FUNCTION_BLOCK PUBLIC ABSTRACT TcoKukaRoboticsTask EXTENDS TcoCore.TcoTask 
VAR_IN_OUT
    inoConfig 	: TcoKukaRobotics_Config_v_5_x_x;
	inoControl 	: TcoKukaRobotics_Control_v_5_x_x;
	inoStatus 	: TcoKukaRobotics_Status_v_5_x_x;	
END_VAR
VAR
	_errorMessage:TcoCore.TcoMessenger(THIS^);
    {attribute 'hide'} 
	_progress : INT := 0;
    {attribute 'hide'} 
	_infoTimer :  TON;
    {attribute 'hide'} 
	_errorTimer :  TON;
	{attribute 'hide'} 
	_timer :  TON;
    {attribute 'hide'} 
	_varInfo : __SYSTEM.VAR_INFO;
    {attribute 'hide'} 
	_sb : TcoCore.StringBuilder;
	{attribute 'hide'}
	_blink:TcoUtilities.TcoBlinker(THIS^);
END_VAR

METHOD CallTimers
VAR_INPUT
	inValue : BOOL;
END_VAR
IF  __ISVALIDREF(inoConfig) AND THIS^.inoConfig.ErrorTime <> T#0S OR NOT inValue THEN  
_errorTimer(IN := inValue, PT := THIS^.inoConfig.ErrorTime);
END_IF;
IF  __ISVALIDREF(inoConfig) AND THIS^.inoConfig.InfoTime <>T#0S OR NOT inValue THEN  
_infoTimer(IN := inValue, PT := THIS^.inoConfig.InfoTime);
END_IF;
END_METHOD

(*~
	<docu>
		<summary>
			Restores this instance to the Ready state. Can be called explicitly or from within one of the restore mechanisms.
			<para>
				See also <see cref="PlcDocu.TcoCore.TcoTask.AutoRestorable()"/>
			</para>
		</summary>			
	</docu>	
~*)
METHOD Restore : ITcoRestorable
SUPER^.Restore();
_progress := 0;
_timer(In:=FALSE);
CallTimers(FALSE);
Messenger.UnPin();
_errorMessage.UnPin();
END_METHOD

END_FUNCTION_BLOCK

(* stored: Version 1.1.0.1, ProductVersion 3.1.4024.12
   POU TcoKukaRoboticsTask: Id {c4d8d758-0a6b-006c-2e1c-ea60ce064bb6}, SpecialFunc None
   Method CallTimers: Id {dd3abd15-d751-0838-3135-8c9a4990f77d}
   Method Restore: Id {4042e357-2a58-0ae9-20bf-c9482f37c624} *)
